# EPICS substitutions: asubtest-mk-IOCApp/Db/userHost3.substitutions
# Example substitutions file

#file "db/asub.db" {
#    { user = "mrippaHost" }
#
#}

file db/asub3.db {
    pattern { user, nsamples, scan }
        { "sim3", 800, "1 second" }
}
